FUNCTION_BLOCK Linearachse
VAR_INPUT
END_VAR
VAR_OUTPUT
END_VAR
VAR
END_VAR

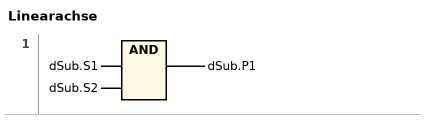
// NETWORK 1
dSub.P1 := dSub.S1 AND dSub.S2;

END_FUNCTION_BLOCK

(* stored: Version 1.1.0.1, ProductVersion 3.1.4022.6
   POU Linearachse: Id {3114a163-c196-4be2-ab35-6259f5e7c1b4}, SpecialFunc None *)
